(* IEC 61131-3 sources: AXOpen/src/integrations/ctrl/src/Examples/ix-core-IxSequencer, 2 files *)

(* ---- IxSequencerDocuExample.st ---- *)
USING AXOpen.Core;

NAMESPACE IxSequencerExamples
    CLASS IxSequencerDocuExample EXTENDS  AXOpen.Core.IxContext
        VAR PUBLIC
            _mySequencer : IxSequencer;
            _step_1 : IxStep;
            _step_2 : IxStep;
            _step_3 : IxStep;
            _myCounter : ULINT;
        END_VAR

    //<Initialize>
        METHOD PUBLIC Initialize
            _mySequencer.Initialize(THIS);
            _step_1.Initialize(THIS);
            _step_2.Initialize(THIS);
            _step_3.Initialize(THIS);
        END_METHOD
    //</Initialize>

        METHOD PROTECTED OVERRIDE Main
    //<Open>
            _mySequencer.Open();
    //</Open>

    //<SimpleStep>
            IF _step_1.Execute(_mySequencer) THEN
                // do something
                _myCounter := _myCounter + ULINT#1;
                IF (_myCounter MOD ULINT#5) = ULINT#0 THEN
                    // continue to the next step of the sequence
                    _mySequencer.MoveNext();
                END_IF;
            END_IF;
    //</SimpleStep>

    //<EnableStep>
            IF _step_2.Execute(coord := _mySequencer, Enable := _myCounter <= ULINT#20) THEN
                _myCounter := _myCounter + ULINT#1;
                IF _myCounter = ULINT#20 THEN
                    // Jumping to step 1. As it is jumping backwards, the execution of step 1
                    // is going to be started in the next context cycle.
                    _mySequencer.RequestStep(_step_1);
                END_IF;
            END_IF;
    //</EnableStep>

   //<FullStep>
            IF _step_3.Execute(coord := _mySequencer, Enable := TRUE, Description := 'This is a description of the step 3' ) THEN
                _myCounter := _myCounter + ULINT#1;
                IF (_myCounter MOD ULINT#7) = ULINT#0 THEN
                    // Finalize the sequence and initiate the execution from the first step.
                    _mySequencer.CompleteSequence();
                END_IF;
            END_IF;
   //</FullStep>
        END_METHOD

    END_CLASS
END_NAMESPACE

(* ---- IxSequencerExample.st ---- *)
USING AXOpen.Core;

NAMESPACE IxSequencerExamples

    CLASS SequencerExample EXTENDS  AXOpen.Core.IxContext
        VAR PUBLIC
            {#ix-set:AttributeName = "<#Sequencer example#>"}
            coord : IxSequencer;
            Counter : ULINT;
        END_VAR

        VAR PUBLIC
            {#ix-set:Description = "Step number one"}
            step_1 : IxStep;
            {#ix-set:Description = "Step number two"}
            step_2 : IxStep;
            {#ix-set:Description = "Step number three"}
            step_3 : IxStep;
            {#ix-set:Description = "Step number four"}
            step_4 : IxStep;
            {#ix-set:Description = "Step number five"}
            step_5 : IxStep;
            {#ix-set:Description = "Step number six"}
            step_6 : IxStep;
            {#ix-set:Description = "Step number seven"}
            step_7 : IxStep;
            {#ix-set:Description = "Step number eight"}
            step_8 : IxStep;
            {#ix-set:Description = "Step number nine"}
            step_9 : IxStep;
            {#ix-set:Description = "Step number ten"}
            step_10 : IxStep;
        END_VAR

        METHOD PROTECTED OVERRIDE Main
            step_1.Initialize(THIS);
            step_2.Initialize(THIS);
            step_3.Initialize(THIS);
            step_4.Initialize(THIS);
            step_5.Initialize(THIS);
            step_6.Initialize(THIS);
            step_7.Initialize(THIS);
            step_8.Initialize(THIS);
            step_9.Initialize(THIS);
            step_10.Initialize(THIS);
            coord.Initialize(THIS);

            coord.Open();

            IF(step_1.Execute(coord)) THEN
                Counter := Counter + ULINT#1;
                IF(Counter >= ULINT#100) THEN
                    Counter := ULINT#0;
                    coord.MoveNext();
                END_IF;
            END_IF;

            IF(step_2.Execute(coord)) THEN
                Counter := Counter + ULINT#1;
                IF(Counter >= ULINT#100) THEN
                    Counter := ULINT#0;
                    coord.MoveNext();
                END_IF;
            END_IF;

            IF(step_3.Execute(coord)) THEN
                Counter := Counter + ULINT#1;
                IF(Counter >= ULINT#100) THEN
                    Counter := ULINT#0;
                    step_3.ThrowWhen(TRUE);
                    coord.MoveNext();
                END_IF;
            END_IF;

            IF(step_4.Execute(coord)) THEN
                Counter := Counter + ULINT#1;
                IF(Counter >= ULINT#100) THEN
                    Counter := ULINT#0;
                    coord.MoveNext();
                END_IF;
            END_IF;

            IF(step_5.Execute(coord)) THEN
                Counter := Counter + ULINT#1;
                IF(Counter >= ULINT#100) THEN
                    Counter := ULINT#0;
                    coord.MoveNext();
                END_IF;
            END_IF;

            IF(step_6.Execute(coord)) THEN
                Counter := Counter + ULINT#1;
                IF(Counter >= ULINT#100) THEN
                    Counter := ULINT#0;
                    coord.MoveNext();
                END_IF;
            END_IF;

            IF(step_7.Execute(coord)) THEN
                Counter := Counter + ULINT#1;
                IF(Counter >= ULINT#100) THEN
                    Counter := ULINT#0;
                    coord.MoveNext();
                END_IF;
            END_IF;

            IF(step_8.Execute(coord)) THEN
                Counter := Counter + ULINT#1;
                IF(Counter >= ULINT#100) THEN
                    Counter := ULINT#0;
                    coord.MoveNext();
                END_IF;
            END_IF;

            IF(step_9.Execute(coord)) THEN
                Counter := Counter + ULINT#1;
                IF(Counter >= ULINT#100) THEN
                    Counter := ULINT#0;
                    coord.MoveNext();
                END_IF;
            END_IF;

            IF(step_10.Execute(coord)) THEN
                Counter := Counter + ULINT#1;
                IF(Counter >= ULINT#100) THEN
                    Counter := ULINT#0;
                    coord.CompleteSequence();
                END_IF;
            END_IF;
        END_METHOD
END_CLASS
END_NAMESPACE
